TYPE Percent : LREAL;
END_TYPE

(* stored: Version 1.1.0.1, ProductVersion 3.1.4024.12
   DUT Percent: Id {7f722e26-47f4-41f3-9b26-4ce8cabfc971} *)
